TYPE ST_JogParameters :
STRUCT
	lrJogAcceleration		:			LREAL;	//Jog acceleration
	lrJogDeceleration		: 			LREAL;	//Jog deceleration
	lrJogJerkValue			:			LREAL;	//Jog jerk
	lrJogVelocity			:			LREAL;	//Jog velocity
	lrJogLimitPositive		:      		LREAL;  // Jog Positive Torque Limit
	lrJogLimitNegative		:			LREAL;  // Jog Negative Torque Limit
END_STRUCT
END_TYPE

(* stored: Version 1.1.0.1, ProductVersion 3.1.4024.6
   DUT ST_JogParameters: Id {b8e0b231-5a22-49c5-bfce-c35a35b21040} *)
